TYPE E_GasType :
(

	none := 0,
	Neon,
	Argon,
	Krypton,
	Xenon,
    Nitrogen

);
END_TYPE

(* stored: Version 1.1.0.1, ProductVersion 3.1.4022.18
   DUT E_GasType: Id {532e7f83-eaf3-47a9-aec9-3260d1893fee} *)
